// TIA Portal V17 export
// export: Created 2023-12-22T15:08:10.0581289Z, ExportSetting WithDefaults, DisplayName Totally Integrated Automation Portal, DisplayVersion V17, DisplayName TIA Portal Openness, DisplayVersion V17, DisplayName TIA Portal Version Control Interface, DisplayVersion V17, DisplayName STEP 7 Professional, DisplayVersion V17, DisplayName STEP 7 Safety, DisplayVersion V17, DisplayName WinCC Advanced, DisplayVersion V17
DATA_BLOCK "PS_cnt_DB"   // DB12
VERSION : 0.1
// stored: AutoNumber false, DBAccessibleFromOPCUA true, DBAccessibleFromWebserver true, InstanceOfName PS_cnt, InstanceOfType FB
"PS_cnt"
   // VAR_INPUT
   //    SP : Real;
   //    REQ : Int;
   // END_VAR
   // VAR_IN_OUT
   //    cnt : Int;
   // END_VAR
   // VAR RETAIN
   //    Select_CMD : Bool;
   //    Select_Mode : Bool;
   //    Select_PS : Int;
   //    PS_Add_Ready : Bool;
   //    PS_Add_CMD : Bool;
   //    SP_Low : Real;
   //    SP_High { S7_SetPoint := 'True'} : Real := 42.0;
   //    SP_Min { S7_SetPoint := 'True'} : Real := 12.0;
   //    cnt_delta { S7_SetPoint := 'True'} : Real := 0.5;
   //    "Step" : Int;
   //    REQ_cnt : Int;
   //    PS_R_OFF : Int;
   //    PS_R_ON : Int;
   //    pos : Array[0..15] of Bool;
   //    tmp : Array[0..15] of Real;
   //    T_Delay_ON { S7_SetPoint := 'True'} : "Time_M";
   //    T_Delay_OFF { S7_SetPoint := 'True'} : "Time_M";
   // END_VAR
BEGIN
   T_Delay_ON.SP_M := 10;
   T_Delay_ON.SP_S := 0;
   T_Delay_OFF.SP_M := 2;
   T_Delay_OFF.SP_S := 30;
END_DATA_BLOCK
